SUBAPPLICATION GreenWhiteBackground1S (* Hintergrundfarbe (TRUE -> Grün, FALSE -> Weiß) für 1 Objekt *)
  (* Standard: 61499-2 *)
  (* Version 1.0, 2024-01-01, franz *)
  PACKAGE MyLib::sys;
  IMPORT isobus::UT::Q::const::IDs::ID_NULL;
  IMPORT isobus::UT::Q::const::colours;
  IMPORT isobus::UT::Q::types::s1ObjectID;
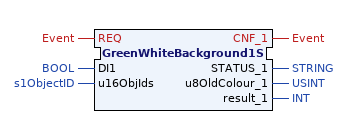
  EVENT_INPUT
    REQ; (* Normal Execution Request *)
  END_EVENT
  EVENT_OUTPUT
    CNF_1; (* Execution Confirmation *)
  END_EVENT
  VAR_INPUT
    DI1 : BOOL; (* Selector *)
    u16ObjIds : isobus::UT::Q::types::s1ObjectID := (u16ObjId := ID_NULL); (* Object IDs *)
  END_VAR
  VAR_OUTPUT
    STATUS_1 : STRING; (* Service Status *)
    u8OldColour_1 : USINT; (* Old value of ID *)
    result_1 : INT; (* retval see description *)
  END_VAR
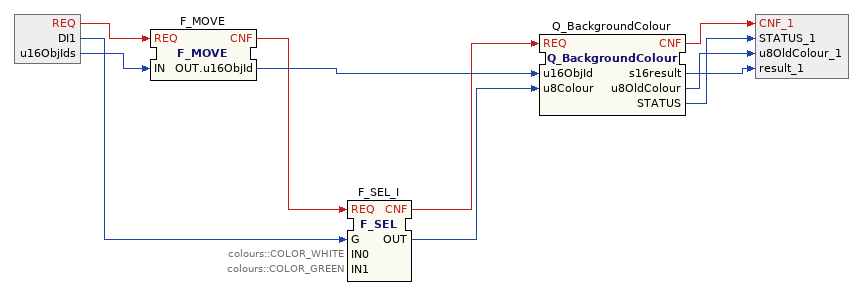
  FBS
    Q_BackgroundColour : isobus::UT::Q::Q_BackgroundColour;
    F_SEL_I : iec61131::selection::F_SEL(IN0 := colours::COLOR_WHITE, IN1 := colours::COLOR_GREEN);
    F_MOVE : iec61131::selection::F_MOVE; {SET_ATTRIBUTE(DataType, isobus::UT::Q::types::s1ObjectID)}
  END_FBS
  EVENT_CONNECTIONS
    Q_BackgroundColour.CNF TO CNF_1;
    F_SEL_I.CNF TO Q_BackgroundColour.REQ;
    REQ TO F_MOVE.REQ;
    F_MOVE.CNF TO F_SEL_I.REQ;
  END_CONNECTIONS
  DATA_CONNECTIONS
    u16ObjIds TO F_MOVE.IN;
    F_MOVE.OUT.u16ObjId TO Q_BackgroundColour.u16ObjId;
    Q_BackgroundColour.s16result TO result_1;
    Q_BackgroundColour.u8OldColour TO u8OldColour_1;
    Q_BackgroundColour.STATUS TO STATUS_1;
    F_SEL_I.OUT TO Q_BackgroundColour.u8Colour;
    DI1 TO F_SEL_I.G;
  END_CONNECTIONS
END_SUBAPPLICATION
